{attribute 'no_explicit_call' := 'do not call this function block directly'} 
// Dynamic dictionary of pointers to key and value
FUNCTION_BLOCK PointerDictionary EXTENDS Object IMPLEMENTS IReadOnlyPointerDictionary
VAR
	_ClassName : STRING := __POUNAME();
	_Keys : POINTER TO PVOID;
	_Values : POINTER TO PVOID;
	_ArrayLength : DINT;
	_ValueCount : DINT;
	_DefaultAllocationElemetsCount : BYTE := 10;
	_KeyType : POINTER_TYPE := POINTER_TYPE.BYTE_POINTER;
	_ValueType : POINTER_TYPE := POINTER_TYPE.BYTE_POINTER;
	_KeyComparer : IPointerComparer;
	_DefaultEnumerator : PointerDictionaryEnumerator;
END_VAR

METHOD AllocateMemory
VAR_INPUT
	elementsCount : DINT;
END_VAR
VAR
	newKeys : POINTER TO PVOID;
	newValues : POINTER TO PVOID;
END_VAR
newKeys := __NEW(PVOID, TO_UDINT(_ArrayLength + elementsCount));
newValues := __NEW(PVOID, TO_UDINT(_ArrayLength + elementsCount));

IF _ValueCount > 0 THEN
	Tc2_System.MEMCPY(newKeys, _Keys, SIZEOF(POINTER TO BYTE) * TO_UDINT(_ValueCount)); 
	Tc2_System.MEMCPY(newValues, _Values, SIZEOF(POINTER TO BYTE) * TO_UDINT(_ValueCount));
END_IF

IF _Keys <> 0 THEN
	__DELETE(_Keys);
END_IF

IF _Values <> 0 THEN
	__DELETE(_Values);
END_IF
 
_Keys := newKeys;
_Values := newValues;
 
_ArrayLength := _ArrayLength + elementsCount;
END_METHOD

{attribute 'monitoring' := 'call'}
PROPERTY ClassName : STRING
GET
ClassName := _ClassName;
END_GET
END_PROPERTY

METHOD Clear
VAR_INPUT
	deleteKeys : BOOL;
	deleteValues : BOOL;
END_VAR
VAR
	i : DINT;
	value : PVOID;
END_VAR
IF deleteKeys AND_THEN _ValueCount > 0 THEN
	FOR i := 0 TO _ValueCount - 1 DO
		TwinCAT_OpenFramework_Core.DynamicMemoryManager.ReleaseDynamicMemory(_Keys[i], _KeyType = POINTER_TYPE.OBJECT_POINTER);						
	END_FOR	
END_IF

IF deleteValues AND_THEN _ValueCount > 0 THEN
	FOR i := 0 TO _ValueCount - 1 DO
		TwinCAT_OpenFramework_Core.DynamicMemoryManager.ReleaseDynamicMemory(_Values[i], _ValueType = POINTER_TYPE.OBJECT_POINTER);
	END_FOR	
END_IF

IF _Keys <> 0 THEN
	__DELETE(_Keys);
END_IF

IF _Values <> 0 THEN
	__DELETE(_Values);
END_IF

_ValueCount := 0;
_ArrayLength := 0;
END_METHOD

METHOD ContainsKey : BOOL
VAR_INPUT
	key : PVOID;
END_VAR
VAR
	index : DINT; 
END_VAR
ContainsKey := SearchKeyPosition(key, supposedIndex => index);
END_METHOD

{attribute 'OPC.UA.DA.Property' := '1'}
{attribute 'monitoring' := 'call'}
PROPERTY Count : DINT
GET
Count := _ValueCount;
END_GET
END_PROPERTY

METHOD FB_exit : BOOL
VAR_INPUT
	bInCopyCode : BOOL; // if TRUE, the exit method is called for exiting an instance that is copied afterwards (online change).
END_VAR
Clear(FALSE, FALSE);
END_METHOD

METHOD FB_init : BOOL
VAR_INPUT
	bInitRetains : BOOL; // if TRUE, the retain variables are initialized (warm start / cold start)
	bInCopyCode : BOOL; // if TRUE, the instance afterwards gets moved into the copy code (online change)
	keyType : POINTER_TYPE;
	valueType : POINTER_TYPE;
	keyComparer : IPointerComparer;
END_VAR
_DefaultEnumerator.Initialize(THIS^);

_KeyType := keyType;
_ValueType := valueType;

IF keyComparer = 0 THEN
	_KeyComparer := StandardPointerComparers.GetForType(keyType);
ELSE
	_KeyComparer := keyComparer;
END_IF
END_METHOD

METHOD GetDefaultEnumerator : IPointerEnumerator
GetDefaultEnumerator := _DefaultEnumerator;
END_METHOD

METHOD GetKeyByIndex : PVOID
VAR_INPUT
	index : DINT;
END_VAR
IF index >= 0 AND index < _ValueCount THEN
	GetKeyByIndex := _Keys[index];
END_IF
END_METHOD

METHOD GetValueByIndex : PVOID
VAR_INPUT
	index : DINT;
END_VAR
IF index >= 0 AND index < _ValueCount THEN
	GetValueByIndex := _Values[index];
END_IF
END_METHOD

METHOD GetValueByKey : PVOID
VAR_INPUT
	key : PVOID;
END_VAR
VAR
	index : DINT; 
END_VAR
IF SearchKeyPosition(key, supposedIndex => index) THEN
	GetValueByKey := _Values[index];
END_IF
END_METHOD

{attribute 'OPC.UA.DA.Property' := '1'}
{attribute 'monitoring' := 'call'}
PROPERTY KeyType : POINTER_TYPE
GET
KeyType := _KeyType;
END_GET
END_PROPERTY

METHOD Remove : BOOL
VAR_INPUT
	key : PVOID;
	deleteKey : BOOL;
	deleteValue : BOOL;
END_VAR
VAR
	index : DINT;
END_VAR
IF SearchKeyPosition(key, supposedIndex => index) THEN
	RemoveAt(index, deleteKey, deleteValue);
	Remove := TRUE;
END_IF
END_METHOD

METHOD RemoveAt : BOOL
VAR_INPUT
	index : DINT;
	deleteKey : BOOL;
	deleteValue : BOOL;
END_VAR
VAR
	i : DINT;
END_VAR
IF index < _ValueCount THEN
	IF deleteKey THEN
		TwinCAT_OpenFramework_Core.DynamicMemoryManager.ReleaseDynamicMemory(_Keys[index], _KeyType = POINTER_TYPE.OBJECT_POINTER);			
	END_IF
	
	IF deleteValue THEN
		TwinCAT_OpenFramework_Core.DynamicMemoryManager.ReleaseDynamicMemory(_Values[index], _ValueType = POINTER_TYPE.OBJECT_POINTER);			
	END_IF
	
	IF index + 2 <= _ValueCount THEN
		FOR	i := index TO _ValueCount - 2 DO
			_Keys[i] := _Keys[i + 1];
			_Values[i] := _Values[i + 1];
		END_FOR			
	END_IF
		
	_Keys[_ValueCount - 1] := 0;
	_Values[_ValueCount - 1] := 0;
	_ValueCount := _ValueCount - 1;
	
	RemoveAt := TRUE;
END_IF
END_METHOD

METHOD PROTECTED SearchKeyPosition : BOOL
VAR_INPUT
	key : PVOID;
END_VAR
VAR_OUTPUT
	supposedIndex : DINT; 
END_VAR
VAR
	lastIndex : DINT;
	minIndex : DINT;
	maxIndex : DINT;
END_VAR
IF _ValueCount = 0 THEN
	RETURN;
END_IF

lastIndex := _ValueCount - 1;
maxIndex := lastIndex;
supposedIndex := maxIndex / 2;

WHILE minIndex <= maxIndex DO
	CASE _KeyComparer.Compare(_Keys[supposedIndex], key) OF
		// assumed key equals to seached 
		COMPARISION_RESULT.FIRST_EQUAL_TO_SECOND:
			SearchKeyPosition := TRUE;
			RETURN;

		// assumed key less than searched, move range to right
		COMPARISION_RESULT.FIRST_LESS_THAN_SECOND:
			minIndex := supposedIndex + 1;
			
		// assumed key greater than searched, move range to left	
		COMPARISION_RESULT.FIRST_GREATER_THAN_SECOND:
			maxIndex := supposedIndex - 1;
	END_CASE
	
	supposedIndex := minIndex + (maxIndex - minIndex) / 2;
END_WHILE
END_METHOD

METHOD Set : DINT
VAR_INPUT
	key : PVOID;
	value : PVOID;
	deleteReplacedKey : BOOL;
	deleteReplacedValue : BOOL;
END_VAR
VAR
	index, i : DINT;
END_VAR
// if equal key found then we need to replace it
IF SearchKeyPosition(key, supposedIndex => index) THEN	
	// old and new keys show to diffirent address, then we need to replace existing key 
	IF _Keys[index] <> key THEN
		IF deleteReplacedKey THEN
			TwinCAT_OpenFramework_Core.DynamicMemoryManager.ReleaseDynamicMemory(_Keys[index], _KeyType = POINTER_TYPE.OBJECT_POINTER);
		END_IF
		
		_Keys[index] := key;
	END_IF
	
	// old and new values show to diffirent address, then we need to replace existing value 
	IF _Values[index] <> value THEN
		IF deleteReplacedValue THEN
			TwinCAT_OpenFramework_Core.DynamicMemoryManager.ReleaseDynamicMemory(_Values[index], _ValueType = POINTER_TYPE.OBJECT_POINTER);
		END_IF
		
		_Values[index] := value;
	END_IF
// if equal key not found than we need to insert it
ELSE
	IF _ValueCount >= _ArrayLength THEN
		AllocateMemory(_DefaultAllocationElemetsCount);
	END_IF
	
	i := _ValueCount;	
	_ValueCount := _ValueCount + 1;
		
	WHILE i > index DO
		_Keys[i] := _Keys[i - 1];
		_Values[i] := _Values[i - 1];
		
		i := i - 1;
	END_WHILE
	
	_Keys[index] := key;
	_Values[index] := value;
END_IF

Set := index;
END_METHOD

{attribute 'monitoring' := 'call'}
PROPERTY Size : ULINT
GET
Size := XSIZEOF(THIS^);
END_GET
END_PROPERTY

{attribute 'OPC.UA.DA.Property' := '1'}
{attribute 'monitoring' := 'call'}
PROPERTY ValueType : POINTER_TYPE
GET
ValueType := _ValueType;
END_GET
END_PROPERTY

END_FUNCTION_BLOCK

(* stored: Version 1.1.0.1
   POU PointerDictionary: Id {1672eefd-21b2-063c-2f9b-b11d951f0d98}, SpecialFunc None
   Method AllocateMemory: Id {8781a493-94d4-0a09-2e01-8d57022ae973}
   Property ClassName: Id {2d52220a-26f8-0028-0278-37e5deeb8d78}
   Get Get: Id {5c789a72-d13b-005e-10aa-40596423b3ff}
   Method Clear: Id {bf9e464d-a2d9-07a3-1cb0-5850ea0c0d6d}
   Method ContainsKey: Id {5e9d864f-5795-0d86-364d-7fee4169a4ed}
   Property Count: Id {03d0cbd5-ff72-00dd-131d-9d17b5aac9e6}
   Get Get: Id {efe807cd-cef9-05d5-02ce-794f47556bbd}
   Method FB_exit: Id {3ce2a3de-ab91-0d2a-2dc4-9e125cca59a0}
   Method FB_init: Id {c6a6e748-9a26-04a7-370f-d370aba5f107}
   Method GetDefaultEnumerator: Id {3cd9f080-5ccc-0a3a-07a6-f62bd5d43e42}
   Method GetKeyByIndex: Id {5b432675-ed86-0ac9-1310-430ec829327f}
   Method GetValueByIndex: Id {bef0986b-7121-0e7f-297f-c38a28387002}
   Method GetValueByKey: Id {4ea24f57-8822-01b2-0147-a148106bf14b}
   Property KeyType: Id {97bb179c-2966-05a4-1c11-c9d76adf254b}
   Get Get: Id {6cb9df5e-9f18-0667-3115-46cb0442e09c}
   Method Remove: Id {6182ced6-3f01-0fd4-37ae-924bbcb45951}
   Method RemoveAt: Id {29c923c9-f082-084d-3a5a-bc3fb1c7fe81}
   Method SearchKeyPosition: Id {dd97240a-5809-08ff-13e6-65d8d9ddf2bb}
   Method Set: Id {41083eda-e38a-08d7-03c2-27b6c8269b9d}
   Property Size: Id {a54786cc-01a6-4a70-887f-ed82cdde2233}
   Get Get: Id {1eb88d76-98f0-4c68-9e66-03fae3cb1b35}
   Property ValueType: Id {e961b863-4945-0050-3bb4-d068ff4b9009}
   Get Get: Id {ab49ed63-427e-0a12-32db-52818d341a65} *)
